// TIA Portal V18 export
// export: Created 2025-12-01T17:51:24.9006127Z, ExportSetting None, DisplayName Totally Integrated Automation Portal, DisplayVersion V18 Update 5, DisplayName TIA Portal Openness, DisplayVersion V18 Update 5, DisplayName TIA Portal Teamcenter Gateway, DisplayVersion V18, DisplayName TIA Portal Version Control Interface, DisplayVersion V18, DisplayName STEP 7 Professional, DisplayVersion V18 Update 5, DisplayName STEP 7 Safety, DisplayVersion V18, DisplayName WinCC Professional, DisplayVersion V18 Update 5
FUNCTION_BLOCK "NGStatus"   // FB2900, LAD
{ S7_Optimized_Access := 'TRUE' }
// stored: AutoNumber false, MemoryReserve 100, SetENOAutomatically false
   VAR_INPUT
      NG_1 : Bool;
      NG_2 : Bool;
      NG_3 : Bool;
      NG_4 : Bool;
      NG_5 : Bool;
   END_VAR
   VAR_OUTPUT
      Status : Int;
      Ready : Bool;
   END_VAR
   VAR_IN_OUT
      Interlock : Array[1..10] of Bool;
   END_VAR
   VAR
      AlwaysOn : Bool;
      NG_Delay : Array[1..10] of TON_TIME;
      NG_DelayTime { S7_SetPoint := 'True'} : Array[1..10] of DInt;
   END_VAR
   // NG_DelayTime[1..10] := 1000;
BEGIN

REGION Network 1: #AlwaysOn
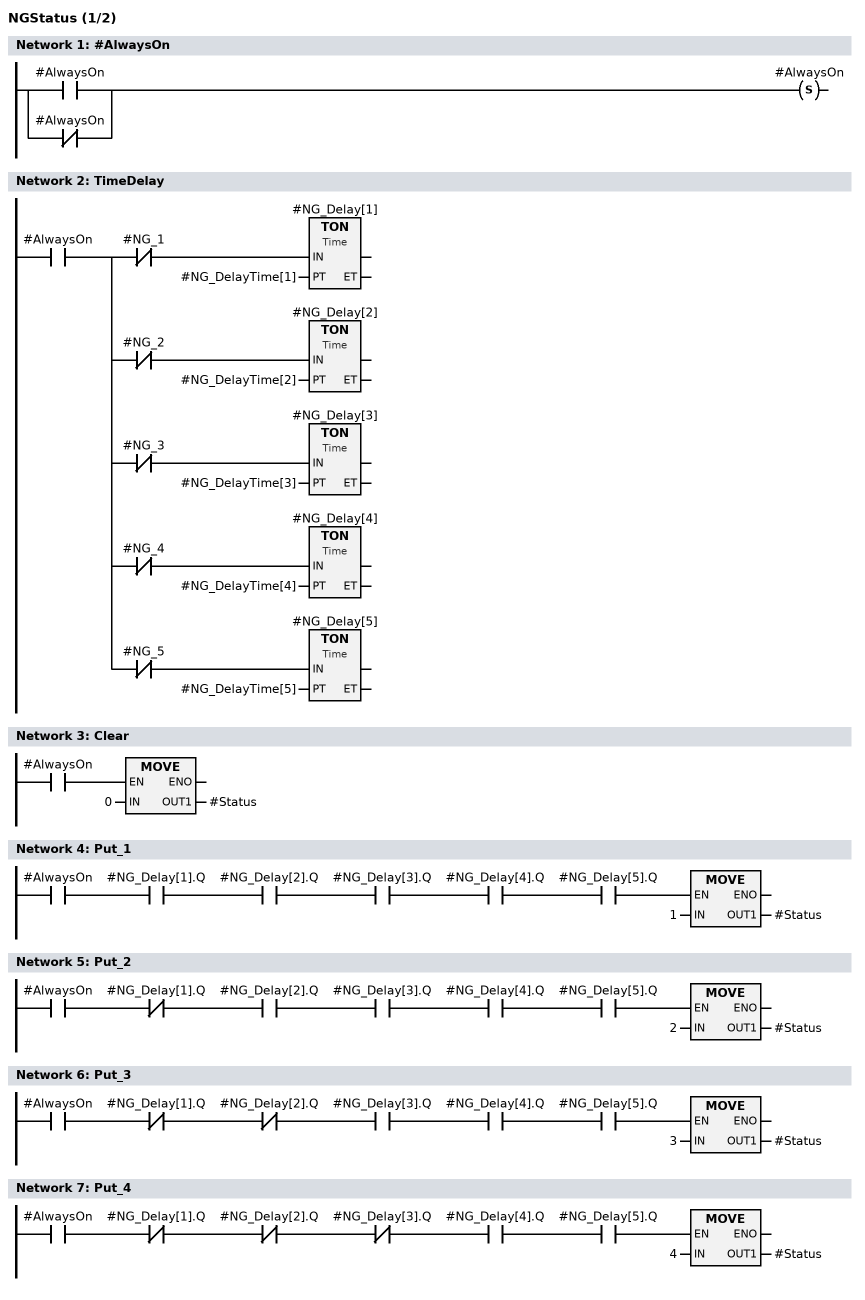
   RUNG wire#powerrail
      Contact( #AlwaysOn )
      wire#w1
      S_Coil( #AlwaysOn )
   END_RUNG
   RUNG wire#powerrail
      I_Contact( #AlwaysOn )
   END_RUNG wire#w1
   // the same network as SCL:
   IF #AlwaysOn OR NOT #AlwaysOn THEN #AlwaysOn := TRUE; END_IF;
END_REGION

REGION Network 2: TimeDelay
   RUNG wire#powerrail
      Contact( #AlwaysOn )
      wire#w1
      I_Contact( #NG_1 )
      { S7_Templates := "time_type := Time" } #NG_Delay[1].TON(pt := #NG_DelayTime[1], et =>)
   END_RUNG
   RUNG wire#w1
      I_Contact( #NG_2 )
      { S7_Templates := "time_type := Time" } #NG_Delay[2].TON(pt := #NG_DelayTime[2], et =>)
   END_RUNG
   RUNG wire#w1
      I_Contact( #NG_3 )
      { S7_Templates := "time_type := Time" } #NG_Delay[3].TON(pt := #NG_DelayTime[3], et =>)
   END_RUNG
   RUNG wire#w1
      I_Contact( #NG_4 )
      { S7_Templates := "time_type := Time" } #NG_Delay[4].TON(pt := #NG_DelayTime[4], et =>)
   END_RUNG
   RUNG wire#w1
      I_Contact( #NG_5 )
      { S7_Templates := "time_type := Time" } #NG_Delay[5].TON(pt := #NG_DelayTime[5], et =>)
   END_RUNG
   // the same network as SCL:
   #NG_Delay[1].TON(IN := #AlwaysOn AND NOT #NG_1, PT := #NG_DelayTime[1]);
   #NG_Delay[2].TON(IN := #AlwaysOn AND NOT #NG_2, PT := #NG_DelayTime[2]);
   #NG_Delay[3].TON(IN := #AlwaysOn AND NOT #NG_3, PT := #NG_DelayTime[3]);
   #NG_Delay[4].TON(IN := #AlwaysOn AND NOT #NG_4, PT := #NG_DelayTime[4]);
   #NG_Delay[5].TON(IN := #AlwaysOn AND NOT #NG_5, PT := #NG_DelayTime[5]);
END_REGION

REGION Network 3: Clear
   RUNG wire#powerrail
      Contact( #AlwaysOn )
      Move(in := 0, out1 => #Status)
   END_RUNG
   // the same network as SCL:
   IF #AlwaysOn THEN #Status := 0; END_IF;
END_REGION

REGION Network 4: Put_1
   RUNG wire#powerrail
      Contact( #AlwaysOn )
      Contact( #NG_Delay[1].Q )
      Contact( #NG_Delay[2].Q )
      Contact( #NG_Delay[3].Q )
      Contact( #NG_Delay[4].Q )
      Contact( #NG_Delay[5].Q )
      Move(in := 1, out1 => #Status)
   END_RUNG
   // the same network as SCL:
   IF #AlwaysOn AND #NG_Delay[1].Q AND #NG_Delay[2].Q AND #NG_Delay[3].Q AND #NG_Delay[4].Q AND #NG_Delay[5].Q THEN
       #Status := 1;
   END_IF;
END_REGION

REGION Network 5: Put_2
   RUNG wire#powerrail
      Contact( #AlwaysOn )
      I_Contact( #NG_Delay[1].Q )
      Contact( #NG_Delay[2].Q )
      Contact( #NG_Delay[3].Q )
      Contact( #NG_Delay[4].Q )
      Contact( #NG_Delay[5].Q )
      Move(in := 2, out1 => #Status)
   END_RUNG
   // the same network as SCL:
   IF #AlwaysOn AND NOT #NG_Delay[1].Q AND #NG_Delay[2].Q AND #NG_Delay[3].Q AND #NG_Delay[4].Q AND #NG_Delay[5].Q THEN
       #Status := 2;
   END_IF;
END_REGION

REGION Network 6: Put_3
   RUNG wire#powerrail
      Contact( #AlwaysOn )
      I_Contact( #NG_Delay[1].Q )
      I_Contact( #NG_Delay[2].Q )
      Contact( #NG_Delay[3].Q )
      Contact( #NG_Delay[4].Q )
      Contact( #NG_Delay[5].Q )
      Move(in := 3, out1 => #Status)
   END_RUNG
   // the same network as SCL:
   IF #AlwaysOn AND NOT #NG_Delay[1].Q AND NOT #NG_Delay[2].Q AND #NG_Delay[3].Q AND #NG_Delay[4].Q AND #NG_Delay[5].Q THEN
       #Status := 3;
   END_IF;
END_REGION

REGION Network 7: Put_4
   RUNG wire#powerrail
      Contact( #AlwaysOn )
      I_Contact( #NG_Delay[1].Q )
      I_Contact( #NG_Delay[2].Q )
      I_Contact( #NG_Delay[3].Q )
      Contact( #NG_Delay[4].Q )
      Contact( #NG_Delay[5].Q )
      Move(in := 4, out1 => #Status)
   END_RUNG
   // the same network as SCL:
   IF #AlwaysOn AND NOT #NG_Delay[1].Q AND NOT #NG_Delay[2].Q AND NOT #NG_Delay[3].Q AND #NG_Delay[4].Q AND #NG_Delay[5].Q THEN
       #Status := 4;
   END_IF;
END_REGION

REGION Network 8: Put_5
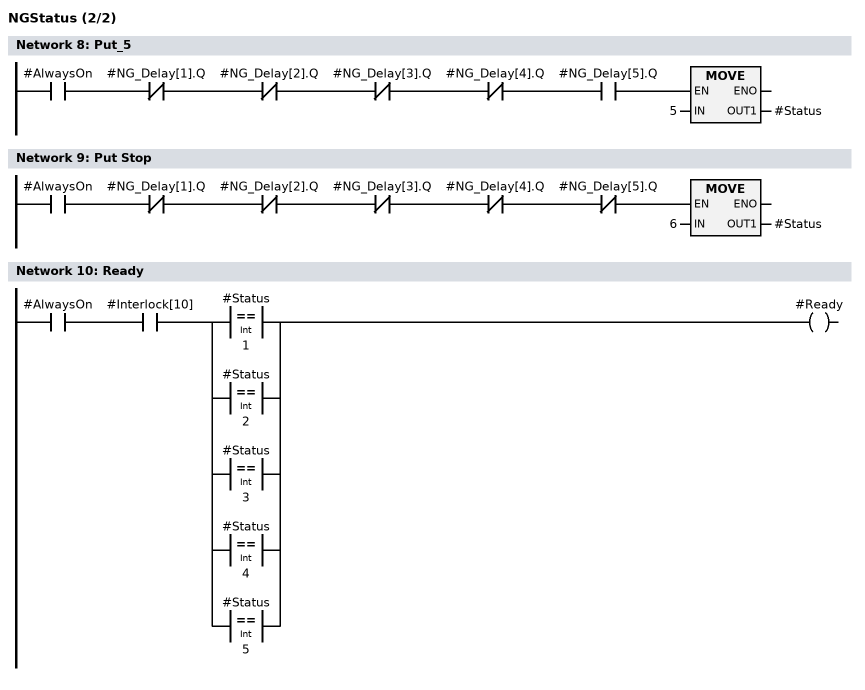
   RUNG wire#powerrail
      Contact( #AlwaysOn )
      I_Contact( #NG_Delay[1].Q )
      I_Contact( #NG_Delay[2].Q )
      I_Contact( #NG_Delay[3].Q )
      I_Contact( #NG_Delay[4].Q )
      Contact( #NG_Delay[5].Q )
      Move(in := 5, out1 => #Status)
   END_RUNG
   // the same network as SCL:
   IF #AlwaysOn AND NOT #NG_Delay[1].Q AND NOT #NG_Delay[2].Q AND NOT #NG_Delay[3].Q AND NOT #NG_Delay[4].Q AND #NG_Delay[5].Q THEN
       #Status := 5;
   END_IF;
END_REGION

REGION Network 9: Put Stop
   RUNG wire#powerrail
      Contact( #AlwaysOn )
      I_Contact( #NG_Delay[1].Q )
      I_Contact( #NG_Delay[2].Q )
      I_Contact( #NG_Delay[3].Q )
      I_Contact( #NG_Delay[4].Q )
      I_Contact( #NG_Delay[5].Q )
      Move(in := 6, out1 => #Status)
   END_RUNG
   // the same network as SCL:
   IF #AlwaysOn AND NOT #NG_Delay[1].Q AND NOT #NG_Delay[2].Q AND NOT #NG_Delay[3].Q AND NOT #NG_Delay[4].Q AND NOT #NG_Delay[5].Q THEN
       #Status := 6;
   END_IF;
END_REGION

REGION Network 10: Ready
   RUNG wire#powerrail
      Contact( #AlwaysOn )
      Contact( #Interlock[10] )
      wire#w1
      { S7_Templates := "SrcType := Int" } EQ_Contact(in1 := #Status, in2 := 1)
      wire#w2
      Coil( #Ready )
   END_RUNG
   RUNG wire#w1
      { S7_Templates := "SrcType := Int" } EQ_Contact(in1 := #Status, in2 := 2)
   END_RUNG wire#w2
   RUNG wire#w1
      { S7_Templates := "SrcType := Int" } EQ_Contact(in1 := #Status, in2 := 3)
   END_RUNG wire#w2
   RUNG wire#w1
      { S7_Templates := "SrcType := Int" } EQ_Contact(in1 := #Status, in2 := 4)
   END_RUNG wire#w2
   RUNG wire#w1
      { S7_Templates := "SrcType := Int" } EQ_Contact(in1 := #Status, in2 := 5)
   END_RUNG wire#w2
   // the same network as SCL:
   #Ready := #AlwaysOn AND #Interlock[10] AND ((#Status = 1) OR (#Status = 2) OR (#Status = 3) OR (#Status = 4) OR (#Status = 5));
END_REGION
END_FUNCTION_BLOCK
